FUNCTION_BLOCK B_TIME_CLOCK (* A simple FB with a single algorithm and REQ/CNF pair *)
  (* Standard: 61499-1 *)
  (* Version 0.0, 2016-01-15, 4DIAC-IDE, 4DIAC-Consortium *)
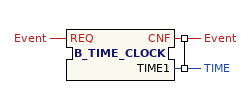
  EVENT_INPUT
    REQ; (* Normal Execution Request *)
  END_EVENT
  EVENT_OUTPUT
    CNF WITH TIME1; (* Execution Confirmation *)
  END_EVENT
  VAR_OUTPUT
    TIME1 : TIME;
  END_VAR
  ALGORITHM REQ IN ST: (* Normally executed algorithm *)
QO := QI;
  END_ALGORITHM
END_FUNCTION_BLOCK
